// TIA Portal V19 export
TYPE "typeStartLift"
TITLE = typeStartLift
// PLC data type start lift
   STRUCT
      startLiftUp : Bool;   // Start lift up
      startLiftDown : Bool;   // Start lift down
   END_STRUCT;
END_TYPE
